Staubli VAL3: Inscribedcircle.pgx

public program Inscribedcircle(trsf& x_trSource[], trsf& x_trCenter, num& x_nDia, bool& x_bRes)
  local num l_ni
  local frame l_fFrame
  local point l_pCenter
  local num a
  local num b
  local num c
  local num p
  local num s
  local num r
  local num l_angle
begin
  //由三角形求内切圆圆心
  //内切圆圆心
  x_bRes=false
  a=distance(x_trSource[0],x_trSource[1])
  b=distance(x_trSource[1],x_trSource[2])
  c=distance(x_trSource[0],x_trSource[2])
  p=(a+b+c)/2
  s=sqrt(p*(p-a)*(p-b)*(p-c))
  r=s/p
  l_angle=acos((c*c+a*a-b*b)/2/a/c)/2

  if l_angle<0
    return
  endIf


  call SetFrame(x_trSource,l_fFrame,x_bRes)
  if !x_bRes
    return
  endIf

  link(l_pCenter,l_fFrame)
  l_pCenter.trsf={r/tan(l_angle),r,0,0,0,0}
  x_trCenter=position(l_pCenter,world)
  x_nDia=r
end
